Fanuc KAREL source: CA0070.KL

PROGRAM CA0070
%STACKSIZE=65535
%PRIORITY=65535
%NOLOCKGROUP
VAR
G : INTEGER
I : INTEGER
R : REAL
B : BOOLEAN
S : STRING[16]
AI : ARRAY[2] OF INTEGER
AR : ARRAY[2] OF REAL
P : XYZWPR
-- UNRESOLVED DECLARATIONS (source type spelling not recovered)
-- ST : TYPE_0x1100 (type_u16=0x1100)
-- V : TYPE_0x0013 (type_u16=0x0013)
ROUTINE F(P1 : INTEGER; P2 : INTEGER; P3 : INTEGER; P4 : INTEGER; P5 : INTEGER; P6 : INTEGER; P7 : INTEGER; P8 : INTEGER; P9 : INTEGER; P10 : INTEGER; P11 : INTEGER; P12 : INTEGER; P13 : INTEGER; P14 : INTEGER; P15 : INTEGER; P16 : INTEGER;
P17 : INTEGER; P18 : INTEGER; P19 : INTEGER; P20 : INTEGER; P21 : INTEGER; P22 : INTEGER; P23 : INTEGER; P24 : INTEGER; P25 : INTEGER; P26 : INTEGER; P27 : INTEGER; P28 : INTEGER; P29 : INTEGER; P30 : INTEGER;
P31 : INTEGER; P32 : INTEGER) FROM CA0070
ROUTINE F
BEGIN
G=(G + 1)
END F
BEGIN
G=0
I=1
R=2.5
B=TRUE
S='A'
AI[1]=3
AR[1]=4.5
ST.A=5
ST.B=1087373312
-- UNSAFE_SOURCE_IR line 64: F(I, ARG_2_UNRESOLVED, I, ARG_4_UNRESOLVED, I, ARG_6_UNRESOLVED, I, ARG_8_UNRESOLVED, I, ARG_10_UNRESOLVED, I, ARG_12_UNRESOLVED, I, ARG_14_UNRESOLVED, I, ARG_16_UNRESOLVED, I, ARG_18_UNRESOLVED, I,
END CA0070
